// TIA Portal V16 export
// export: Created 2024-09-05T17:39:12.465902Z, ExportSetting WithDefaults, DisplayName Totally Integrated Automation Portal, DisplayVersion V16 Update 6, DisplayName TIA Portal Version Control Interface, DisplayVersion V16 Update 2, DisplayName TIA Portal Openness, DisplayVersion V16 Update 6, DisplayName STEP 7 Professional, DisplayVersion V16 Update 6, DisplayName STEP 7 Safety, DisplayVersion V16, DisplayName WinCC Advanced, DisplayVersion V16 Update 6
DATA_BLOCK "RivetingHistoryRight_DB"   // DB23
VERSION : 0.1
// stored: AutoNumber true, DBAccessibleFromOPCUA true, InstanceOfName RivetingHistory, InstanceOfType FB
"RivetingHistory"
   // VAR_INPUT
   //    iNewCycle : Bool;
   //    iData : "UDT_Friedrich";
   // END_VAR
   // VAR RETAIN
   //    history : Array[0..99] of "UDT_Friedrich";
   // END_VAR
   // VAR
   //    pageData { S7_SetPoint := 'True'} : Array[0..9] of "UDT_Friedrich";
   // END_VAR
   // VAR RETAIN
   //    pageNumber { S7_SetPoint := 'True'} : USInt := 0;
   // END_VAR
   // VAR
   //    resetHistory : Bool;
   // END_VAR
BEGIN
   history[0..99].Start := FALSE;
   history[0..24].PrgNumber := 2;
   history[25..52].PrgNumber := 1;
   history[53..66].PrgNumber := 2;
   history[67].PrgNumber := 1;
   history[68..99].PrgNumber := 0;
   history[0..11].Ready := TRUE;
   history[12].Ready := FALSE;
   history[13..67].Ready := TRUE;
   history[68..99].Ready := FALSE;
   history[0..99].Running := FALSE;
   history[0..19].OK := TRUE;
   history[20..22].OK := FALSE;
   history[23].OK := TRUE;
   history[24].OK := FALSE;
   history[25..32].OK := TRUE;
   history[33].OK := FALSE;
   history[34..35].OK := TRUE;
   history[36].OK := FALSE;
   history[37..43].OK := TRUE;
   history[44..99].OK := FALSE;
   history[0..19].NOK := FALSE;
   history[20..22].NOK := TRUE;
   history[23].NOK := FALSE;
   history[24].NOK := TRUE;
   history[25..32].NOK := FALSE;
   history[33].NOK := TRUE;
   history[34..35].NOK := FALSE;
   history[36].NOK := TRUE;
   history[37..43].NOK := FALSE;
   history[44..67].NOK := TRUE;
   history[68..99].NOK := FALSE;
   history[0..32].H1OK := TRUE;
   history[33].H1OK := FALSE;
   history[34..35].H1OK := TRUE;
   history[36].H1OK := FALSE;
   history[37..55].H1OK := TRUE;
   history[56..99].H1OK := FALSE;
   history[0..19].H2OK := TRUE;
   history[20..22].H2OK := FALSE;
   history[23].H2OK := TRUE;
   history[24].H2OK := FALSE;
   history[25..32].H2OK := TRUE;
   history[33].H2OK := FALSE;
   history[34..35].H2OK := TRUE;
   history[36].H2OK := FALSE;
   history[37..43].H2OK := TRUE;
   history[44..99].H2OK := FALSE;
   history[0..23].TimeOK := TRUE;
   history[24].TimeOK := FALSE;
   history[25..32].TimeOK := TRUE;
   history[33].TimeOK := FALSE;
   history[34..35].TimeOK := TRUE;
   history[36].TimeOK := FALSE;
   history[37..43].TimeOK := TRUE;
   history[44..99].TimeOK := FALSE;
   history[0..99].StartError := FALSE;
   history[0..24].LastH1 := 0.0;
   history[25].LastH1 := 5.09;
   history[26].LastH1 := 5.17;
   history[27].LastH1 := 5.11;
   history[28].LastH1 := 5.29;
   history[29].LastH1 := 5.23;
   history[30].LastH1 := 5.18;
   history[31].LastH1 := 5.22;
   history[32].LastH1 := 5.0;
   history[33].LastH1 := 4.84;
   history[34].LastH1 := 5.27;
   history[35].LastH1 := 5.26;
   history[36].LastH1 := -0.11;
   history[37].LastH1 := 5.25;
   history[38].LastH1 := 2.47;
   history[39..99].LastH1 := 0.0;
   history[0..3].LastH2 := 0.0;
   history[4].LastH2 := 2.37;
   history[5..6].LastH2 := 2.38;
   history[7..8].LastH2 := 2.4;
   history[9].LastH2 := 2.39;
   history[10].LastH2 := 2.38;
   history[11].LastH2 := 2.4;
   history[12..13].LastH2 := 2.39;
   history[14].LastH2 := 0.19;
   history[15].LastH2 := 2.39;
   history[16..17].LastH2 := 0.19;
   history[18].LastH2 := 0.18;
   history[19].LastH2 := 0.19;
   history[20].LastH2 := 0.18;
   history[21].LastH2 := 0.19;
   history[22].LastH2 := 0.18;
   history[23].LastH2 := 2.37;
   history[24].LastH2 := 0.0;
   history[25..26].LastH2 := 2.38;
   history[27].LastH2 := 2.36;
   history[28].LastH2 := 2.4;
   history[29].LastH2 := 2.39;
   history[30].LastH2 := 2.38;
   history[31].LastH2 := 2.33;
   history[32].LastH2 := 2.38;
   history[33].LastH2 := 0.0;
   history[34].LastH2 := 2.4;
   history[35].LastH2 := 2.39;
   history[36].LastH2 := 0.0;
   history[37].LastH2 := 2.39;
   history[38].LastH2 := 2.4;
   history[39].LastH2 := 2.39;
   history[40].LastH2 := 2.4;
   history[41].LastH2 := 2.38;
   history[42].LastH2 := 2.39;
   history[43].LastH2 := 2.4;
   history[44..99].LastH2 := 0.0;
   history[0..3].LastTime := 0.0;
   history[4].LastTime := 1.47;
   history[5].LastTime := 0.96;
   history[6].LastTime := 0.98;
   history[7].LastTime := 0.65;
   history[8].LastTime := 0.68;
   history[9].LastTime := 1.01;
   history[10].LastTime := 0.94;
   history[11].LastTime := 0.86;
   history[12..13].LastTime := 0.15;
   history[14].LastTime := 0.0;
   history[15].LastTime := 0.33;
   history[16..22].LastTime := 0.0;
   history[23].LastTime := 0.83;
   history[24].LastTime := 0.0;
   history[25].LastTime := 1.94;
   history[26].LastTime := 2.55;
   history[27].LastTime := 2.14;
   history[28].LastTime := 2.35;
   history[29].LastTime := 2.7;
   history[30].LastTime := 2.31;
   history[31].LastTime := 2.17;
   history[32].LastTime := 2.47;
   history[33].LastTime := 0.0;
   history[34].LastTime := 2.34;
   history[35].LastTime := 2.88;
   history[36].LastTime := 0.0;
   history[37].LastTime := 2.21;
   history[38].LastTime := 0.12;
   history[39].LastTime := 2.58;
   history[40].LastTime := 2.51;
   history[41].LastTime := 2.3;
   history[42].LastTime := 2.34;
   history[43].LastTime := 2.54;
   history[44..99].LastTime := 0.0;
   history[0].LastZ1 := 11.96;
   history[1].LastZ1 := 12.01;
   history[2].LastZ1 := 12.11;
   history[3].LastZ1 := 12.1;
   history[4].LastZ1 := 12.38;
   history[5..6].LastZ1 := 12.2;
   history[7].LastZ1 := 12.14;
   history[8].LastZ1 := 12.13;
   history[9].LastZ1 := 12.19;
   history[10].LastZ1 := 12.0;
   history[11].LastZ1 := 12.18;
   history[12..13].LastZ1 := 12.58;
   history[14].LastZ1 := 12.33;
   history[15].LastZ1 := 12.6;
   history[16].LastZ1 := 12.34;
   history[17].LastZ1 := 12.33;
   history[18].LastZ1 := 12.32;
   history[19..20].LastZ1 := 12.3;
   history[21].LastZ1 := 12.33;
   history[22].LastZ1 := 12.3;
   history[23..24].LastZ1 := 12.43;
   history[25].LastZ1 := 15.42;
   history[26].LastZ1 := 15.4;
   history[27].LastZ1 := 15.41;
   history[28].LastZ1 := 15.4;
   history[29].LastZ1 := 15.39;
   history[30].LastZ1 := 15.4;
   history[31].LastZ1 := 15.39;
   history[32].LastZ1 := 15.42;
   history[33].LastZ1 := 15.43;
   history[34].LastZ1 := 15.41;
   history[35].LastZ1 := 15.44;
   history[36].LastZ1 := 8.43;
   history[37].LastZ1 := 15.42;
   history[38].LastZ1 := 12.39;
   history[39].LastZ1 := 15.39;
   history[40].LastZ1 := 15.46;
   history[41].LastZ1 := 15.42;
   history[42].LastZ1 := 15.43;
   history[43].LastZ1 := 15.39;
   history[44].LastZ1 := 13.18;
   history[45..47].LastZ1 := 13.2;
   history[48].LastZ1 := 3.22;
   history[49..99].LastZ1 := 0.0;
   history[0..99].Error := FALSE;
   history[0..99].NewData := FALSE;
   history[0..23].Z1OK := TRUE;
   history[24].Z1OK := FALSE;
   history[25..35].Z1OK := TRUE;
   history[36].Z1OK := FALSE;
   history[37..43].Z1OK := TRUE;
   history[44..99].Z1OK := FALSE;
   history[0..48].NewDataAfterStart := TRUE;
   history[49..99].NewDataAfterStart := FALSE;
   history[0].LastZ2 := 11.96;
   history[1].LastZ2 := 12.01;
   history[2].LastZ2 := 12.11;
   history[3].LastZ2 := 12.1;
   history[4..99].LastZ2 := 0.0;
END_DATA_BLOCK
